Yaskawa INFORM job: R1_W17,20,22(0,0)OK-KMNEW2.JBI

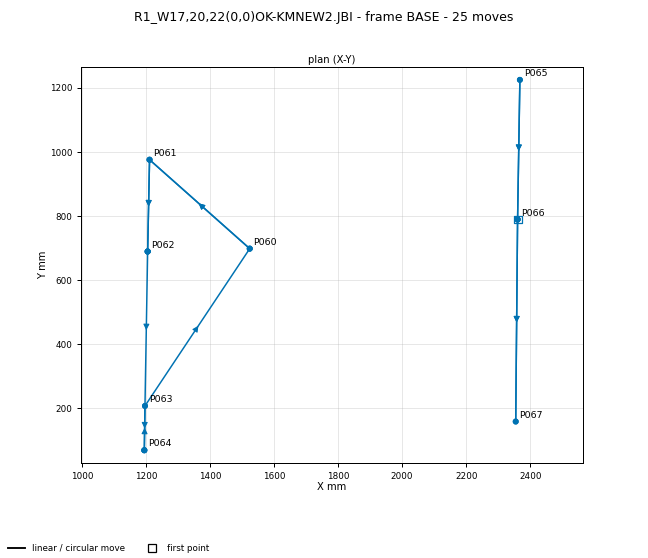
[picture p0: tool path of R1_W17,20,22(0,0)OK-KMNEW2.JBI in frame BASE, 25 of 140 moves have a stored position in this frame; points joined in program order, loops and branches not executed]
/JOB
//NAME R1_W17,20,22(0,0)OK-KMNEW2
///FOLDERNAME KRIS-SCIANA
//POS
///NPOS 83,83,0,12,0,0
///TOOL 0
///POSTYPE PULSE
///PULSE
C00000=-143433,-90175,-75020,-14586,83972,33032
C00001=-157098,-74863,-52692,-13875,75874,29154
C00002=-157098,-74532,-51903,-13892,75569,29189
C00003=-157098,-74863,-52692,-13875,75874,29154
C00004=-211231,-128371,-70027,-7339,52125,11439
C00005=-211231,-127849,-69381,-7351,51997,11448
C00006=-211231,-128371,-70027,-7339,52125,11439
C00007=-232444,-131211,-70558,-2415,49804,3169
C00008=-232444,-130212,-69358,-2423,49579,3175
C00009=-232444,-131211,-70558,-2415,49804,3169
C00010=-132869,-107414,-81260,-15133,81051,37100
C00011=-145969,-32332,-29442,-14415,85137,32009
C00012=-145969,-32299,-29299,-14416,85068,32017
C00013=-145969,-32158,-28695,-14420,84777,32051
C00014=-145969,-32299,-29299,-14416,85068,32017
C00015=-139425,14349,7377,-14755,87604,34007
C00016=-139425,14458,7934,-14756,87328,34041
C00017=-139425,14349,7377,-14755,87604,34007
C00018=-140402,1849,-19527,-14902,97240,32509
C00019=-140435,1808,-19560,-14885,97235,32499
C00020=-142735,11930,7018,-14580,86016,33037
C00021=-142735,12166,8091,-14585,85494,33098
C00022=-142735,11930,7018,-14580,86016,33037
C00023=-153871,-49427,-38150,-13936,80432,29777
C00024=-153871,-49122,-37171,-13951,80000,29826
C00025=-153871,-49427,-38150,-13936,80432,29777
C00026=-177115,-82244,-48475,-26198,85674,24082
C00027=-177115,-82011,-48031,-26200,85536,24113
C00028=-177115,-82244,-48475,-26198,85674,24082
C00029=-152058,-57095,-47355,-15849,91689,31553
C00030=-158551,-98871,-68851,-16167,82483,30472
C00031=-139863,-9121,-22514,-12675,86754,36604
C00032=-142907,-1645,-8358,-12312,81526,36078
C00033=-146433,-61661,-62839,-14679,91621,33634
C00034=-152691,-57358,-64796,-14380,93822,31204
C00035=-159687,-62193,-51187,-13527,81199,28324
C00036=-189185,-159173,-100064,-12251,58132,22119
C00037=-139628,-22178,-29745,-13339,88451,36438
C00038=-142464,16713,5801,-14603,90978,35100
C00039=-142912,-78923,-74681,-14594,91271,34909
C00040=96,-41537,-55485,-8102,54341,61135
C00041=96,-41537,-55485,-8102,54341,61135
C00042=-47991,-26757,-28892,6367,80786,-11975
C00043=-57126,-9114,2182,8032,71615,-15703
C00044=-57153,4111,18055,10725,70923,-22649
C00045=-57153,4533,19124,10752,70490,-22688
C00046=-57153,4111,18055,10725,70923,-22649
C00047=-38989,-22714,-2775,8400,67834,-16383
C00048=-38989,-22525,-2315,8410,67650,-16396
C00049=-38989,-22714,-2775,8400,67834,-16383
C00050=-17967,-38347,-13490,5028,64666,-8942
C00051=-17967,-38006,-12720,5040,64367,-8955
C00052=-17967,-38347,-13490,5028,64666,-8942
C00053=23595,-40752,-17055,-2802,65045,6207
C00054=23156,-37209,-12609,-2742,64116,6069
C00055=23156,-36957,-12035,-2747,63893,6074
C00056=23156,-37209,-12609,-2742,64116,6069
C00057=33691,-30497,-8275,-4656,65373,9871
C00058=33691,-29938,-6960,-4674,64853,9891
C00059=33691,-30497,-8275,-4656,65373,9871
C00060=33691,-40237,-37529,-4343,78333,9389
C00061=4088,-38479,-36421,-4266,78531,9229
C00062=6240,-59965,-30493,-1746,62990,4256
C00063=6240,-59594,-29713,-1750,62700,4261
C00064=5477,-60554,-32035,-1584,63620,3965
C00065=42086,-42798,-20663,-6177,66949,12973
C00066=42086,-42521,-20002,-6189,66686,12987
C00067=42086,-42798,-20663,-6177,66949,12973
C00068=65240,-6064,10187,5043,53635,20347
C00069=65240,-5748,10977,5064,53312,20331
C00070=65240,-6064,10187,5043,53635,20347
C00071=61085,-36100,-21666,6391,58079,18912
C00072=61085,-36100,-21666,6391,58079,18912
C00073=29040,-81101,-50034,-3867,64562,8354
C00074=7217,-74366,-42042,361,62632,377
C00075=46390,-61269,-41061,-6756,70352,14356
C00076=42236,-65961,-43421,-6101,69070,12939
C00077=45032,-34460,-3825,-6892,61383,14260
C00078=78652,23072,35845,-11228,70256,25748
C00079=41637,-60211,-42225,-5828,71489,12454
C00080=-9438,-58348,-23745,3601,60262,-5968
C00081=50643,-51074,-27069,-7729,67873,16514
C00082=-88506,-94181,-91931,-709,81235,59832
BC00000=335653,8129,711615
BC00001=335653,8129,711615
BC00002=335653,8129,711615
BC00003=335653,8129,711615
BC00004=335653,8130,711613
BC00005=335653,8130,711613
BC00006=335653,8130,711613
BC00007=335653,1154,711613
BC00008=335653,1154,711613
BC00009=335653,1154,711613
BC00010=335653,1154,711613
BC00011=335653,1154,711613
BC00012=335653,1154,711613
BC00013=335653,1154,711613
BC00014=335653,1154,711613
BC00015=335653,1152,711610
BC00016=335653,1152,711610
BC00017=335653,1152,711610
BC00018=335653,1152,711610
BC00019=160380,1151,711608
BC00020=160380,1151,715049
BC00021=160380,1151,715049
BC00022=160380,1151,715049
BC00023=160380,1151,715049
BC00024=160380,1151,715049
BC00025=160380,1151,715049
BC00026=160380,1151,715049
BC00027=160380,1151,715049
BC00028=160380,1151,715049
BC00029=160380,1151,715049
BC00030=160381,1151,715048
BC00031=160381,1151,715048
BC00032=160381,1151,715048
BC00033=160381,1151,715048
BC00034=347379,1151,715048
BC00035=347379,1151,715048
BC00036=347379,1151,715048
BC00037=347379,1151,715048
BC00038=347379,1151,715048
BC00039=347379,1151,715048
BC00040=71294,1151,1035267
BC00041=71294,1151,1035267
BC00042=14908,77377,861464
BC00043=14908,77377,833834
BC00044=14908,77377,833834
BC00045=14908,77377,833834
BC00046=14908,77377,833834
BC00047=14908,77377,833834
BC00048=14908,77377,833834
BC00049=14908,77377,833834
BC00050=14908,77377,833834
BC00051=14908,77377,833834
BC00052=14908,77377,833834
BC00053=14908,77377,833834
BC00054=14908,77377,833834
BC00055=14908,77377,833834
BC00056=14908,77377,833834
BC00057=14908,77377,833834
BC00058=14908,77377,833834
BC00059=14908,77377,833834
BC00060=14908,77377,833834
BC00061=166638,196652,833834
BC00062=218128,196652,810863
BC00063=218128,196652,810863
BC00064=218128,196652,810863
BC00065=218128,196652,810863
BC00066=218128,196652,810863
BC00067=218128,196652,810863
BC00068=218128,196652,810863
BC00069=218128,196652,810863
BC00070=218128,196652,810863
BC00071=218128,196652,810863
BC00072=218128,196652,810863
BC00073=218128,196652,810863
BC00074=218128,196652,810863
BC00075=218128,196652,810863
BC00076=35771,188457,887876
BC00077=35771,188457,887876
BC00078=35772,185483,887872
BC00079=35772,185483,887872
BC00080=35772,185483,887872
BC00081=38104,183984,886436
BC00082=294911,15771,909309
///POSTYPE BASE
///RECTAN
///RCONF 0,0,0,0,0,0,0,0,0,0,0,0,0,0,0,0,0,0,0,0,0,0,0,0
P00060=1524.284,698.404,-261.973,-0.4635,36.8346,-1.2388
P00061=1211.499,975.999,-261.374,0.5148,35.2356,175.5099
P00062=1205.574,689.500,-262.704,0.5159,35.2461,175.5270
P00063=1197.217,207.358,-268.729,0.4863,35.2395,175.4586
P00064=1195.199,68.975,-269.171,0.5092,35.2366,175.4908
P00065=2367.684,1225.356,-251.745,0.6375,35.5356,-175.5535
P00066=2360.514,789.486,-255.123,0.6232,35.5414,175.8162
P00067=2354.696,158.615,-258.055,26.2211,34.3929,-169.2888
P00100=-8.801,1.165,-9.977,0.0000,0.0000,0.0000
P00125=0.000,0.000,2.400,0.0000,0.0000,0.0000
P00126=-50.000,0.000,0.000,0.0000,0.0000,0.0000
P00127=50.000,0.000,0.000,0.0000,0.0000,0.0000
//INST
///DATE 2024/07/18 11:13
///ATTR SC,RW
///GROUP1 RB1,BS1
///LVARS 0,1,0,0,0,2,2,0
NOP
MOVJ C00000 BC00000 VJ=50.00
SFTOF
MOVL C00001 BC00001 V=166.7
MOVL C00002 BC00002 V=16.7 SRCH RIN#(1)=ON T=1.00 DIS=40.0
IMOV P125 V=23.0
IMOV P126 V=23.0 SRCH RIN#(1)=ON T=1.00 DIS=40.0
TIMER T=0.10
GETS PX060 $PX001
TIMER T=0.10
MOVL C00003 BC00003 V=166.7
MOVL C00004 BC00004 V=166.7
MOVL C00005 BC00005 V=16.7 SRCH RIN#(1)=ON T=1.00 DIS=40.0
IMOV P125 V=23.0
IMOV P126 V=23.0 SRCH RIN#(1)=ON T=1.00 DIS=40.0
TIMER T=0.10
GETS PX061 $PX001
TIMER T=0.10
MOVL C00006 BC00006 V=166.7
MOVL C00007 BC00007 V=166.7
MOVL C00008 BC00008 V=16.7 SRCH RIN#(1)=ON T=1.00 DIS=40.0
IMOV P125 V=23.0
IMOV P126 V=23.0 SRCH RIN#(1)=ON T=1.00 DIS=40.0
TIMER T=0.10
GETS PX062 $PX001
TIMER T=0.10
MOVL C00009 BC00009 V=166.7
MOVJ C00010 BC00010 VJ=25.00
MOVJ C00011 BC00011 VJ=25.00
MOVL C00012 BC00012 V=166.7
MOVL C00013 BC00013 V=16.7 SRCH RIN#(1)=ON T=1.00 DIS=40.0
IMOV P125 V=23.0
IMOV P126 V=23.0 SRCH RIN#(1)=ON T=1.00 DIS=40.0
TIMER T=0.10
GETS PX063 $PX001
TIMER T=0.10
MOVL C00014 BC00014 V=166.7
MOVL C00015 BC00015 V=166.7
MOVL C00016 BC00016 V=16.7 SRCH RIN#(1)=ON T=1.00 DIS=40.0
IMOV P125 V=23.0
IMOV P126 V=23.0 SRCH RIN#(1)=ON T=1.00 DIS=40.0
TIMER T=0.10
GETS PX064 $PX001
TIMER T=0.10
MOVL C00017 BC00017 V=166.7
MOVL C00018 BC00018 V=166.7
MOVL C00019 BC00019 V=166.7
MOVL C00020 BC00020 V=166.7
MOVL C00021 BC00021 V=16.7 SRCH RIN#(1)=ON T=1.00 DIS=40.0
IMOV P125 V=23.0
IMOV P126 V=23.0 SRCH RIN#(1)=ON T=1.00 DIS=40.0
TIMER T=0.10
GETS PX065 $PX001
TIMER T=0.10
MOVL C00022 BC00022 V=166.7
MOVL C00023 BC00023 V=166.7
MOVL C00024 BC00024 V=16.7 SRCH RIN#(1)=ON T=1.00 DIS=40.0
IMOV P125 V=23.0
IMOV P126 V=23.0 SRCH RIN#(1)=ON T=1.00 DIS=40.0
TIMER T=0.10
GETS PX066 $PX001
TIMER T=0.10
MOVL C00025 BC00025 V=166.7
MOVL C00026 BC00026 V=166.7
MOVL C00027 BC00027 V=16.7 SRCH RIN#(1)=ON T=1.00 DIS=40.0
IMOV P125 V=23.0
IMOV P126 V=23.0 SRCH RIN#(1)=ON T=1.00 DIS=40.0
TIMER T=0.10
GETS PX067 $PX001
TIMER T=0.10
MOVL C00028 BC00028 V=166.7
MOVL C00029 BC00029 V=166.7
MACRO1 MJ#(0) ARGF9
SFTON P100
MOVL P066 V=83.3
ARCON
MOVL P067 V=12.5
ARCOF
SFTOF
MOVJ C00030 BC00030 VJ=25.00
MOVJ C00031 BC00031 VJ=25.00
MOVJ C00032 BC00032 VJ=25.00
MOVL P065 V=83.3
ARCON
SFTON P100
MOVL P066 V=12.5
ARCOF
SFTOF
MOVJ C00033 BC00033 VJ=25.00
MOVJ C00034 BC00034 VJ=25.00
MOVJ C00035 BC00035 VJ=25.00
SFTON P100
MOVL P060 V=83.3
ARCON
MOVL P061 V=10.8
MOVL P061 V=10.8
ARCOF
MOVL P062 V=41.7
SFTOF
ARCON
SFTON P100
MOVL P062 V=10.8
MOVL P062 V=10.8
ARCOF
SFTOF
MOVJ C00036 BC00036 VJ=25.00
MOVJ C00037 BC00037 VJ=25.00
MOVJ C00038 BC00038 VJ=25.00
MOVL P064 V=83.3
ARCON
SFTON P100
MOVL P063 V=10.8
MOVL P060 V=10.8
ARCOF
SFTOF
MOVJ C00039 BC00039 VJ=25.00
MOVJ C00040 BC00040 VJ=25.00
CALL JOB:CLEAN-R1_LONG
MOVJ C00041 BC00041 VJ=25.00
MOVJ C00042 BC00042 VJ=25.00
MOVJ C00043 BC00043 VJ=25.00
MOVL C00044 BC00044 V=166.7
MOVL C00045 BC00045 V=16.7 SRCH RIN#(1)=ON T=1.00 DIS=40.0
IMOV P125 V=23.0
IMOV P127 V=23.0 SRCH RIN#(1)=ON T=1.00 DIS=40.0
TIMER T=0.10
GETS PX060 $PX001
TIMER T=0.10
MOVL C00046 BC00046 V=166.7
MOVL C00047 BC00047 V=166.7
MOVL C00048 BC00048 V=16.7 SRCH RIN#(1)=ON T=1.00 DIS=40.0
IMOV P125 V=23.0
IMOV P127 V=23.0 SRCH RIN#(1)=ON T=1.00 DIS=40.0
TIMER T=0.10
GETS PX061 $PX001
TIMER T=0.10
MOVL C00049 BC00049 V=166.7
MOVL C00050 BC00050 V=166.7
MOVL C00051 BC00051 V=16.7 SRCH RIN#(1)=ON T=1.00 DIS=40.0
IMOV P125 V=23.0
IMOV P127 V=23.0 SRCH RIN#(1)=ON T=1.00 DIS=40.0
TIMER T=0.10
GETS PX062 $PX001
TIMER T=0.10
MOVL C00052 BC00052 V=166.7
MOVL C00053 BC00053 V=250.0
MOVL C00054 BC00054 V=166.7
MOVL C00055 BC00055 V=16.7 SRCH RIN#(1)=ON T=1.00 DIS=40.0
IMOV P125 V=23.0
IMOV P127 V=23.0 SRCH RIN#(1)=ON T=1.00 DIS=40.0
TIMER T=0.10
GETS PX063 $PX001
TIMER T=0.10
MOVL C00056 BC00056 V=166.7
MOVL C00057 BC00057 V=166.7
MOVL C00058 BC00058 V=16.7 SRCH RIN#(1)=ON T=1.00 DIS=40.0
IMOV P125 V=23.0
IMOV P127 V=23.0 SRCH RIN#(1)=ON T=1.00 DIS=40.0
TIMER T=0.10
GETS PX064 $PX001
TIMER T=0.10
MOVL C00059 BC00059 V=166.7
MOVL C00060 BC00060 V=166.7
MOVL C00061 BC00061 V=166.7
MOVL C00062 BC00062 V=166.7
MOVL C00063 BC00063 V=16.7 SRCH RIN#(1)=ON T=1.00 DIS=40.0
IMOV P125 V=23.0
IMOV P127 V=23.0 SRCH RIN#(1)=ON T=1.00 DIS=40.0
TIMER T=0.10
GETS PX065 $PX001
TIMER T=0.10
MOVL C00064 BC00064 V=166.7
MOVL C00065 BC00065 V=166.7
MOVL C00066 BC00066 V=16.7 SRCH RIN#(1)=ON T=1.00 DIS=40.0
IMOV P125 V=23.0
IMOV P127 V=23.0 SRCH RIN#(1)=ON T=1.00 DIS=40.0
TIMER T=0.10
GETS PX066 $PX001
TIMER T=0.10
MOVL C00067 BC00067 V=166.7
MOVL C00068 BC00068 V=166.7
MOVL C00069 BC00069 V=16.7 SRCH RIN#(1)=ON T=1.00 DIS=40.0
IMOV P125 V=23.0
IMOV P127 V=23.0 SRCH RIN#(1)=ON T=1.00 DIS=40.0
TIMER T=0.10
GETS PX067 $PX001
TIMER T=0.10
MOVL C00070 BC00070 V=166.7
MOVL C00071 BC00071 V=166.7
MACRO1 MJ#(0) ARGF9
SFTON P100
MOVL P066 V=83.3
ARCON
MOVL P067 V=12.5
ARCOF
SFTOF
MOVJ C00072 BC00072 VJ=25.00
MOVJ C00073 BC00073 VJ=25.00
MOVJ C00074 BC00074 VJ=25.00
MOVL P065 V=83.3
ARCON
SFTON P100
MOVL P066 V=12.5
ARCOF
SFTOF
MOVJ C00075 BC00075 VJ=25.00
MOVJ C00076 BC00076 VJ=25.00
MOVJ C00077 BC00077 VJ=25.00
SFTON P100
MOVL P062 V=83.3
ARCON
MOVL P063 V=10.8
SFTOF
ARCOF
MOVL P064 V=41.7
SFTOF
SFTON P100
ARCON
MOVL P064 V=10.8
MOVL P064 V=10.0
ARCOF
SFTOF
MOVJ C00078 BC00078 VJ=25.00
MOVJ C00079 BC00079 VJ=25.00
MOVJ C00080 BC00080 VJ=25.00
MOVL P060 V=83.3
ARCON
SFTON P100
MOVL P061 V=10.8
MOVL P062 V=10.8
ARCOF
SFTOF
MOVJ C00081 BC00081 VJ=40.00
MOVJ C00082 BC00082 VJ=40.00
END
